// TIA Portal project "Soru10" (V15)

(* hardware
DEVICE "S7-1200 station_1"  S7-1200 Station
   slot 0: "Rack_0"  S7-1200 Rack  Rack  V1.0
   slot 1: "PLC_1"  CPU 1214C DC/DC/DC  6ES7 214-1AG40-0XB0  V4.2
*)

// ===== PLC "PLC_1"  CPU 1214C DC/DC/DC =====

VAR_GLOBAL   // PLC tag table "Default tag table"
   "Dudur" AT %I0.0 : Bool;
   "Pause" AT %I0.1 : Bool;
   "Baslat" AT %I0.2 : Bool;
   "Motor_1" AT %Q0.0 : Bool;
   "Motor_2" AT %Q0.1 : Bool;
   "Motor_3" AT %Q0.2 : Bool;
   "Motor_4" AT %Q0.3 : Bool;
   "41snDoldu" AT %M0.0 : Bool;
END_VAR

// folder: System blocks/Program resources

DATA_BLOCK "Say"   // DB1
{ S7_Optimized_Access := 'TRUE' }
AUTHOR : Simatic
FAMILY : IEC
NAME : IEC_TMR
VERSION : 1.0
// stored: InstanceOfName IEC_TIMER
"IEC_TIMER"
BEGIN
END_DATA_BLOCK

// folder: (top level)

ORGANIZATION_BLOCK "Main"   // OB1, LAD, ProgramCycle
TITLE = "Main Program Sweep (Cycle)"
{ S7_Optimized_Access := 'TRUE' }
VERSION : 0.1
   VAR_INPUT
      Initial_Call : Bool;   // Initial call of this OB
      Remanence : Bool;   // =True, if remanent data are available
   END_VAR
BEGIN

REGION Network 1: Zaman rölesi
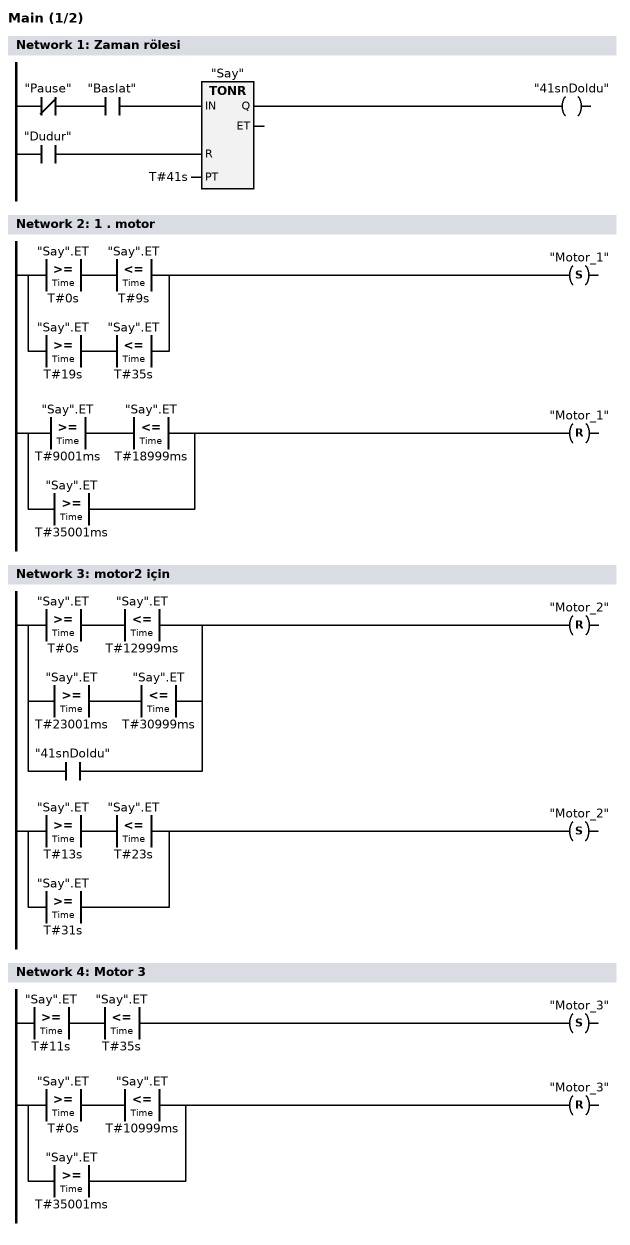
   "Say".TONR(IN := NOT "Pause" AND "Baslat", R := "Dudur", PT := T#41s);
   "41snDoldu" := "Say".Q;
END_REGION

REGION Network 2: 1 . motor
   RUNG wire#powerrail
      { S7_Templates := "SrcType := Time" } GE_Contact(in1 := "Say".ET, in2 := T#0s)
      { S7_Templates := "SrcType := Time" } LE_Contact(in1 := "Say".ET, in2 := T#9s)
      wire#w1
      S_Coil( "Motor_1" )
   END_RUNG
   RUNG wire#powerrail
      { S7_Templates := "SrcType := Time" } GE_Contact(in1 := "Say".ET, in2 := T#19s)
      { S7_Templates := "SrcType := Time" } LE_Contact(in1 := "Say".ET, in2 := T#35s)
   END_RUNG wire#w1
   RUNG wire#powerrail
      { S7_Templates := "SrcType := Time" } GE_Contact(in1 := "Say".ET, in2 := T#9001ms)
      { S7_Templates := "SrcType := Time" } LE_Contact(in1 := "Say".ET, in2 := T#18999ms)
      wire#w2
      R_Coil( "Motor_1" )
   END_RUNG
   RUNG wire#powerrail
      { S7_Templates := "SrcType := Time" } GE_Contact(in1 := "Say".ET, in2 := T#35001ms)
   END_RUNG wire#w2
   // the same network as SCL:
   IF (("Say".ET >= T#0s) AND ("Say".ET <= T#9s)) OR (("Say".ET >= T#19s) AND ("Say".ET <= T#35s)) THEN
       "Motor_1" := TRUE;
   END_IF;
   IF (("Say".ET >= T#9001ms) AND ("Say".ET <= T#18999ms)) OR ("Say".ET >= T#35001ms) THEN
       "Motor_1" := FALSE;
   END_IF;
END_REGION

REGION Network 3: motor2 için
   RUNG wire#powerrail
      { S7_Templates := "SrcType := Time" } GE_Contact(in1 := "Say".ET, in2 := T#0s)
      { S7_Templates := "SrcType := Time" } LE_Contact(in1 := "Say".ET, in2 := T#12999ms)
      wire#w1
      R_Coil( "Motor_2" )
   END_RUNG
   RUNG wire#powerrail
      { S7_Templates := "SrcType := Time" } GE_Contact(in1 := "Say".ET, in2 := T#23001ms)
      { S7_Templates := "SrcType := Time" } LE_Contact(in1 := "Say".ET, in2 := T#30999ms)
   END_RUNG wire#w1
   RUNG wire#powerrail
      Contact( "41snDoldu" )
   END_RUNG wire#w1
   RUNG wire#powerrail
      { S7_Templates := "SrcType := Time" } GE_Contact(in1 := "Say".ET, in2 := T#13s)
      { S7_Templates := "SrcType := Time" } LE_Contact(in1 := "Say".ET, in2 := T#23s)
      wire#w2
      S_Coil( "Motor_2" )
   END_RUNG
   RUNG wire#powerrail
      { S7_Templates := "SrcType := Time" } GE_Contact(in1 := "Say".ET, in2 := T#31s)
   END_RUNG wire#w2
   // the same network as SCL:
   IF (("Say".ET >= T#0s) AND ("Say".ET <= T#12999ms)) OR (("Say".ET >= T#23001ms) AND ("Say".ET <= T#30999ms)) OR "41snDoldu" THEN
       "Motor_2" := FALSE;
   END_IF;
   IF (("Say".ET >= T#13s) AND ("Say".ET <= T#23s)) OR ("Say".ET >= T#31s) THEN "Motor_2" := TRUE; END_IF;
END_REGION

REGION Network 4: Motor 3
   RUNG wire#powerrail
      { S7_Templates := "SrcType := Time" } GE_Contact(in1 := "Say".ET, in2 := T#11s)
      { S7_Templates := "SrcType := Time" } LE_Contact(in1 := "Say".ET, in2 := T#35s)
      S_Coil( "Motor_3" )
   END_RUNG
   RUNG wire#powerrail
      { S7_Templates := "SrcType := Time" } GE_Contact(in1 := "Say".ET, in2 := T#0s)
      { S7_Templates := "SrcType := Time" } LE_Contact(in1 := "Say".ET, in2 := T#10999ms)
      wire#w1
      R_Coil( "Motor_3" )
   END_RUNG
   RUNG wire#powerrail
      { S7_Templates := "SrcType := Time" } GE_Contact(in1 := "Say".ET, in2 := T#35001ms)
   END_RUNG wire#w1
   // the same network as SCL:
   IF ("Say".ET >= T#11s) AND ("Say".ET <= T#35s) THEN "Motor_3" := TRUE; END_IF;
   IF (("Say".ET >= T#0s) AND ("Say".ET <= T#10999ms)) OR ("Say".ET >= T#35001ms) THEN
       "Motor_3" := FALSE;
   END_IF;
END_REGION

REGION Network 5: 4 . motor
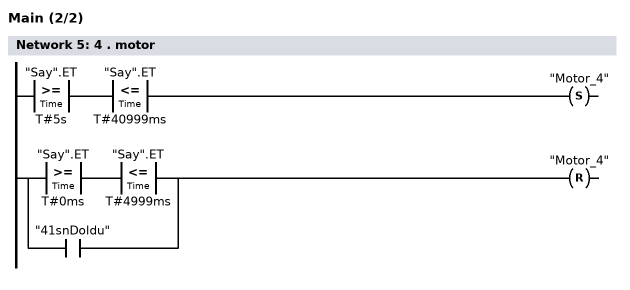
   RUNG wire#powerrail
      { S7_Templates := "SrcType := Time" } GE_Contact(in1 := "Say".ET, in2 := T#5s)
      { S7_Templates := "SrcType := Time" } LE_Contact(in1 := "Say".ET, in2 := T#40999ms)
      S_Coil( "Motor_4" )
   END_RUNG
   RUNG wire#powerrail
      { S7_Templates := "SrcType := Time" } GE_Contact(in1 := "Say".ET, in2 := T#0ms)
      { S7_Templates := "SrcType := Time" } LE_Contact(in1 := "Say".ET, in2 := T#4999ms)
      wire#w1
      R_Coil( "Motor_4" )
   END_RUNG
   RUNG wire#powerrail
      Contact( "41snDoldu" )
   END_RUNG wire#w1
   // the same network as SCL:
   IF ("Say".ET >= T#5s) AND ("Say".ET <= T#40999ms) THEN "Motor_4" := TRUE; END_IF;
   IF (("Say".ET >= T#0ms) AND ("Say".ET <= T#4999ms)) OR "41snDoldu" THEN "Motor_4" := FALSE; END_IF;
END_REGION
END_ORGANIZATION_BLOCK